Staubli VAL3: MotionBuffer.dtx

public mdesc mVelAcc = {leave=0, reach=0}
public num nDuration
public num nSequence
public jointRx jJointRx
